FUNCTION_BLOCK FB_SecondBlock EXTENDS FB_MyBlock
VAR_INPUT
END_VAR
VAR_OUTPUT
END_VAR
VAR
END_VAR

END_FUNCTION_BLOCK

(* stored: Version 1.1.0.1, ProductVersion 3.1.4024.11
   POU FB_SecondBlock: Id {5b1a58fd-6131-41bc-aa58-fd0a19d2321e}, SpecialFunc None *)
